FUNCTION_BLOCK aFb_Valve
VAR_INPUT
	Mode: aE_Mode := aE_Mode.Manual;
	
	//Manual
	Start: BOOL;
	Stop: BOOL;
	SetPercent: REAL;
	Reset1: BOOL;
	
	//Auto
	RunCondition: BOOL;
	StopCondition: BOOL;
	PercentCondition: REAL;
	
	//Others
	RunFeedback: BOOL;
	Interlock: BOOL;
END_VAR
VAR_OUTPUT
	Cmd: BOOL;
	Fault: BOOL;
	State: aE_State;
	OpenPercent: REAL;
	Runtime: UDINT := 0;
	AccRuntime: UDINT := 0;
END_VAR
VAR
	{attribute 'hide'}
	fbTon: TON;
	{attribute 'hide'}
	fbTRuntime: TON;	
END_VAR

CASE Mode OF 
	aE_Mode.Manual: 
		Cmd := (Cmd OR Start) AND NOT Stop AND NOT Fault AND NOT Interlock;
		IF Cmd THEN
			State := aE_State.ManRun;
		ELSE
			State := aE_State.ManStop;
		END_IF
	aE_Mode.Auto:
		Cmd := (Cmd OR RunCondition) AND NOT StopCondition AND NOT Fault AND NOT Interlock;
		State := aE_State.Auto;
	aE_Mode.Service:
		Cmd := (Cmd OR Start) AND NOT Stop AND NOT Fault;
END_CASE

IF Cmd THEN
	IF Mode = aE_Mode.Auto THEN
		OpenPercent := LIMIT( 0, PercentCondition, 1);
	ELSE
		OpenPercent := LIMIT( 0, SetPercent, 1);
	END_IF
ELSE 
	OpenPercent:= 0;
END_IF

fbTon(IN := Cmd, PT := T#3S);
IF fbTon.Q AND NOT RunFeedback THEN
	Fault := TRUE;
	State := aE_State.Fault;
END_IF

IF Reset1 THEN
	Fault := FALSE;
END_IF

IF Cmd THEN
	fbTRuntime(IN := NOT fbTRuntime.Q, PT:= T#1S);
	IF fbTRuntime.Q THEN
		Runtime:= Runtime + 1;
		AccRuntime := AccRuntime + 1;
	END_IF
ELSE
	Runtime:= 0;
END_IF

END_FUNCTION_BLOCK

(* stored: Version 1.1.0.1, ProductVersion 3.1.4024.4
   POU aFB_Valve: Id {3d1810ca-99c6-4a27-a7c3-1ca372238459}, SpecialFunc None *)
